PROGRAM MAIN
VAR
Elevation : FB_Elevation;
Azimuth : FB_Azimuth;
END_VAR

Elevation();
Azimuth();

END_PROGRAM

(* stored: Version 1.1.0.1, ProductVersion 3.1.4024.12
   POU MAIN: Id {d2ef0984-92bd-496a-889d-abe550655014}, SpecialFunc None *)
